// TIA Portal V18 export
// export: Created 2026-06-11T18:57:32.5220549Z, ExportSetting WithDefaults, DisplayName Totally Integrated Automation Portal, DisplayVersion V18, DisplayName TIA Portal Openness, DisplayVersion V18, DisplayName TIA Portal Version Control Interface, DisplayVersion V18, DisplayName STEP 7 Professional, DisplayVersion V18, DisplayName STEP 7 Safety, DisplayVersion V18, DisplayName WinCC Professional, DisplayVersion V18
Screen "scadabai3"  1920x1080, Number=4
  ScreenLayer 
    GraphicView "Graphic view_1" at 0,-1 size 1924x1081  Picture=21a25079-727b-40d3-bd7b-d97467a50c1b
    Button "Button_1" at 419,20 size 129x36  Mode=Text, TextOff="Press1 priority", TextOn="Text"
    Button "Button_2" at 558,20 size 124x37  Mode=Text, TextOff="Press2 priority", TextOn="Text"
    Button "Button_3" at 700,24 size 182x33  Mode=Text, TextOff="CIP PSC MODE", TextOn="Text"
    IOField "I/O field_1" at 41,55 size 141x31  DataFormat=Decimal, FormatPattern=99999999, Mode=InOutput
    Button "Button_6" at 420,57 size 262x36  Mode=Text, TextOff="Press1", TextOn="Text"
    IOField "I/O field_2" at 227,242 size 42x28  DataFormat=Decimal, FormatPattern=99999999, Mode=InOutput
    IOField "I/O field_3" at 462,239 size 46x33  DataFormat=Decimal, FormatPattern=99999999, Mode=InOutput
    IOField "I/O field_4" at 535,256 size 43x29  DataFormat=Decimal, FormatPattern=99999999, Mode=InOutput
    IOField "I/O field_5" at 531,191 size 44x29  DataFormat=Decimal, FormatPattern=99999999, Mode=InOutput
    Circle "Circle_1" at 734,251 size 22x22
    IOField "I/O field_6" at 1076,147 size 66x28  DataFormat=Decimal, FormatPattern=99999999, Mode=InOutput
    IOField "I/O field_7" at 1174,416 size 47x33  DataFormat=Decimal, FormatPattern=99999999, Mode=InOutput
    IOField "I/O field_8" at 49,357 size 47x35  DataFormat=Decimal, FormatPattern=99999999, Mode=InOutput
    IOField "I/O field_9" at 353,416 size 44x28  DataFormat=Decimal, FormatPattern=99999999, Mode=InOutput
    IOField "I/O field_10" at 112,586 size 45x32  DataFormat=Decimal, FormatPattern=99999999, Mode=InOutput
    IOField "I/O field_11" at 202,599 size 48x34  DataFormat=Decimal, FormatPattern=99999999, Mode=InOutput
    IOField "I/O field_12" at 317,837 size 43x27  DataFormat=Decimal, FormatPattern=99999999, Mode=InOutput
    IOField "I/O field_13" at 383,835 size 45x29  DataFormat=Decimal, FormatPattern=99999999, Mode=InOutput
    IOField "I/O field_14" at 224,915 size 45x28  DataFormat=Decimal, FormatPattern=99999999, Mode=InOutput
    IOField "I/O field_15" at 277,930 size 43x29  DataFormat=Decimal, FormatPattern=99999999, Mode=InOutput
    IOField "I/O field_16" at 383,930 size 46x29  DataFormat=Decimal, FormatPattern=99999999, Mode=InOutput
    IOField "I/O field_17" at 443,930 size 44x28  DataFormat=Decimal, FormatPattern=99999999, Mode=InOutput
    IOField "I/O field_18" at 609,745 size 49x36  DataFormat=Decimal, FormatPattern=99999999, Mode=InOutput
    IOField "I/O field_19" at 866,743 size 47x33  DataFormat=Decimal, FormatPattern=99999999, Mode=InOutput
    IOField "I/O field_20" at 992,800 size 47x33  DataFormat=Decimal, FormatPattern=99999999, Mode=InOutput
    IOField "I/O field_21" at 866,904 size 43x28  DataFormat=Decimal, FormatPattern=99999999, Mode=InOutput
    IOField "I/O field_22" at 937,943 size 43x28  DataFormat=Decimal, FormatPattern=99999999, Mode=InOutput
    IOField "I/O field_23" at 942,994 size 46x28  DataFormat=Decimal, FormatPattern=99999999, Mode=InOutput
    IOField "I/O field_24" at 1006,994 size 50x28  DataFormat=Decimal, FormatPattern=99999999, Mode=InOutput
    IOField "I/O field_25" at 1280,871 size 47x33  DataFormat=Decimal, FormatPattern=99999999, Mode=InOutput
    IOField "I/O field_26" at 1423,871 size 47x33  DataFormat=Decimal, FormatPattern=99999999, Mode=InOutput
    IOField "I/O field_27" at 1595,864 size 47x33  DataFormat=Decimal, FormatPattern=99999999, Mode=InOutput
    IOField "I/O field_28" at 1834,864 size 47x33  DataFormat=Decimal, FormatPattern=99999999, Mode=InOutput
    IOField "I/O field_29" at 419,466 size 47x36  DataFormat=Decimal, FormatPattern=99999999, Mode=InOutput
    IOField "I/O field_30" at 169,270 size 42x28  DataFormat=Decimal, FormatPattern=99999999, Mode=InOutput
    IOField "I/O field_31" at 1497,730 size 44x28  DataFormat=Decimal, FormatPattern=99999999, Mode=InOutput
    IOField "I/O field_32" at 1672,729 size 44x28  DataFormat=Decimal, FormatPattern=99999999, Mode=InOutput
    IOField "I/O field_33" at 1781,728 size 42x27  DataFormat=Decimal, FormatPattern=99999999, Mode=InOutput
    IOField "I/O field_34" at 1781,809 size 41x25  DataFormat=Decimal, FormatPattern=99999999, Mode=InOutput
    Rectangle "Rectangle_1" at 105,787 size 12x13
    Rectangle "Rectangle_2" at 74,703 size 14x13
    Rectangle "Rectangle_3" at 343,713 size 14x13
    GraphicView "Graphic view_2" at 1126,726 size 49x39  Picture=d1ddbce5-8e7f-4e40-850e-34ecdf8c874e
    Circle "Circle_2" at 91,491 size 25x25
    Circle "Circle_3" at 124,106 size 15x15
    Circle "Circle_4" at 182,187 size 10x10
    Circle "Circle_5" at 217,196 size 11x11
    Circle "Circle_6" at 264,195 size 10x10
    Circle "Circle_7" at 295,203 size 10x10
    Circle "Circle_8" at 360,187 size 10x10
    Circle "Circle_9" at 397,194 size 10x10
    Circle "Circle_10" at 204,329 size 10x10
    Circle "Circle_11" at 91,537 size 10x10
    Circle "Circle_12" at 214,1031 size 23x23
    Circle "Circle_13" at 286,1031 size 23x23
    Circle "Circle_14" at 358,1017 size 26x26
    Circle "Circle_15" at 412,1031 size 23x23
    Circle "Circle_16" at 451,1031 size 23x23
    Circle "Circle_17" at 518,1022 size 26x26
    Circle "Circle_18" at 571,1031 size 23x23
    Circle "Circle_19" at 1213,951 size 25x25
    Circle "Circle_20" at 1213,992 size 26x26
    Circle "Circle_21" at 1470,989 size 26x26
    Circle "Circle_22" at 1648,986 size 26x26
    Circle "Circle_23" at 1787,845 size 30x30
    TextField "Text field_1" at 1797,849 size 12x21  Text="R"
    Circle "Circle_24" at 1680,765 size 30x30
    TextField "Text field_2" at 1690,770 size 12x21  Text="R"
    Circle "Circle_25" at 376,547 size 10x10
    Circle "Circle_26" at 394,547 size 10x10
    Circle "Circle_27" at 572,601 size 10x10
    Circle "Circle_28" at 589,601 size 10x10
    Circle "Circle_29" at 604,601 size 10x10
    Circle "Circle_30" at 532,648 size 10x10
    Circle "Circle_31" at 544,648 size 10x10
    Circle "Circle_32" at 561,648 size 10x10
    Circle "Circle_33" at 336,658 size 10x10
    Circle "Circle_34" at 320,658 size 10x10
    Circle "Circle_35" at 768,691 size 14x14
    Circle "Circle_36" at 524,690 size 14x14
    Circle "Circle_37" at 544,571 size 11x11
    Circle "Circle_38" at 506,623 size 11x11
    Button "Button_4" at 683,786 size 54x29  Mode=Text, TextOff="REV", TextOn="Text"
    Button "Button_5" at 738,785 size 54x29  Mode=Text, TextOff="PWO", TextOn="Text"
    Circle "Circle_39" at 746,897 size 10x10
    Circle "Circle_40" at 1007,260 size 14x14
    Circle "Circle_41" at 1263,262 size 14x14
    Circle "Circle_42" at 1202,449 size 10x10
    Circle "Circle_43" at 1253,519 size 11x11
    Circle "Circle_44" at 1269,519 size 11x11
    Circle "Circle_45" at 1638,534 size 10x10
    Circle "Circle_46" at 1653,534 size 10x10
    Rectangle "Rectangle_4" at 165,101 size 14x11
    Rectangle "Rectangle_5" at 102,180 size 14x11
    Rectangle "Rectangle_6" at 230,279 size 10x9
    Rectangle "Rectangle_7" at 230,309 size 11x9
    Rectangle "Rectangle_8" at 224,363 size 14x9
    Rectangle "Rectangle_9" at 345,379 size 14x10
    Rectangle "Rectangle_10" at 444,381 size 14x10
    Rectangle "Rectangle_11" at 444,424 size 15x8
    Rectangle "Rectangle_12" at 379,516 size 15x8
    Rectangle "Rectangle_13" at 502,514 size 8x16
    Rectangle "Rectangle_14" at 538,514 size 8x16
    Rectangle "Rectangle_15" at 580,515 size 9x15
    Rectangle "Rectangle_16" at 584,667 size 17x9
    Rectangle "Rectangle_17" at 311,656 size 7x15
    Rectangle "Rectangle_18" at 169,517 size 15x8
    Rectangle "Rectangle_19" at 177,638 size 15x10
    Rectangle "Rectangle_20" at 206,829 size 15x10
    Rectangle "Rectangle_21" at 258,854 size 15x12
    Rectangle "Rectangle_22" at 472,874 size 8x17
    Rectangle "Rectangle_23" at 548,899 size 14x10
    Rectangle "Rectangle_24" at 715,899 size 7x15
    Rectangle "Rectangle_26" at 967,806 size 14x14
    Rectangle "Rectangle_27" at 1101,850 size 10x18
    Rectangle "Rectangle_28" at 1084,900 size 16x8
    Bar "Bar_1" at 1333,843 size 8x72  CountSubDivisions=2, IntegerDigits=2, LargeTickLabelingStep=1, MaximumValue=5, MinimumValue=-5, Precision=2
    Bar "Bar_2" at 1474,843 size 9x73  CountSubDivisions=2, IntegerDigits=2, LargeTickLabelingStep=1, MaximumValue=5, MinimumValue=-5, Precision=2
    Bar "Bar_3" at 1644,843 size 9x72  CountSubDivisions=2, IntegerDigits=2, LargeTickLabelingStep=1, MaximumValue=5, MinimumValue=-5, Precision=2
    Bar "Bar_4" at 1889,841 size 10x74  CountSubDivisions=2, IntegerDigits=2, LargeTickLabelingStep=1, MaximumValue=5, MinimumValue=-5, Precision=2
    Bar "Bar_5" at 339,416 size 12x130  CountSubDivisions=2, IntegerDigits=2, LargeTickLabelingStep=1, MaximumValue=5, MinimumValue=-5, Precision=2
    Rectangle "Rectangle_29" at 307,130 size 17x9
    Rectangle "Rectangle_30" at 342,130 size 16x9
    Rectangle "Rectangle_31" at 650,170 size 16x10
    Rectangle "Rectangle_32" at 754,171 size 11x16
    Rectangle "Rectangle_33" at 910,223 size 10x15
    Rectangle "Rectangle_34" at 1011,222 size 10x16
    Rectangle "Rectangle_35" at 1168,223 size 10x15
    Rectangle "Rectangle_36" at 1267,223 size 11x16
    Rectangle "Rectangle_37" at 1294,178 size 9x16
    Rectangle "Rectangle_38" at 1377,178 size 10x15
    Rectangle "Rectangle_39" at 1436,177 size 11x16
    Rectangle "Rectangle_40" at 1463,177 size 10x16
    Rectangle "Rectangle_41" at 1598,175 size 10x18
    Rectangle "Rectangle_42" at 1628,177 size 10x16
    Rectangle "Rectangle_43" at 1658,428 size 11x10
    Circle "Circle_47" at 1628,516 size 10x10
    Rectangle "Rectangle_44" at 1624,529 size 12x18
    Rectangle "Rectangle_45" at 1848,593 size 8x18
    Rectangle "Rectangle_46" at 1859,685 size 15x11
    Rectangle "Rectangle_47" at 1242,517 size 10x17
    Rectangle "Rectangle_48" at 1246,502 size 9x12
    Circle "Circle_48" at 1187,466 size 10x10
    Circle "Circle_49" at 1167,298 size 27x27
    Circle "Circle_50" at 915,298 size 27x27
    Circle "Circle_51" at 436,250 size 14x14
    Circle "Circle_52" at 102,367 size 14x14
    Button "Button_7" at 1504,240 size 30x35  Mode=Text, TextOff="Text", TextOn="Text"
    Button "Button_8" at 1674,242 size 30x35  Mode=Text, TextOff="Text", TextOn="Text"
    Circle "Circle_53" at 1502,765 size 31x31
    TextField "Text field_3" at 1514,770 size 12x21  Text="R"
    TextField "Text field_4" at 768,487 size 168x38  Text="Lien Gia Bao"
    Rectangle "Rectangle_49" at 1144,721 size 17x10
    Rectangle "Rectangle_50" at 838,620 size 17x13
    Rectangle "Rectangle_51" at 838,662 size 17x13
    Rectangle "Rectangle_52" at 162,595 size 15x10
    Rectangle "Rectangle_53" at 254,604 size 15x10
    Rectangle "Rectangle_54" at 954,870 size 16x9
    Rectangle "Rectangle_55" at 942,840 size 14x9
    Circle "Circle_54" at 924,872 size 25x25
    Circle "Circle_55" at 910,875 size 12x12
    Circle "Circle_56" at 726,898 size 12x12
    Button "Button_9" at 712,331 size 33x40  Mode=Text, TextOff="Text", TextOn="Text"
    Button "Btn_Enter_System_4" at 1806,0 size 114x38  Mode=Text, StyleItem=Button, TextOff="Mh login", TextOn="Text"
      VisibilityAnimation "VisibilityAnimation"  RangeEnd=99, RangeStart=1
        tag Logged_In
      on Click: ActivateScreen(Screen name := Login/out, Object number := 0)
